# EPICS autosave request: iocBoot/sioc-cha-bkhM1/bkhM1.req
file ../bkhMot.req P=$(P),MOT=2531-1,M=$(M)
